FUNCTION_BLOCK DoorControl (* Basic Function Block Type *)
  (* Standard: 61499-2 *)
  (* Version 0.0, 6/17/2016, Andrei, nxtControl GmbH, Template *)
  PACKAGE Main;
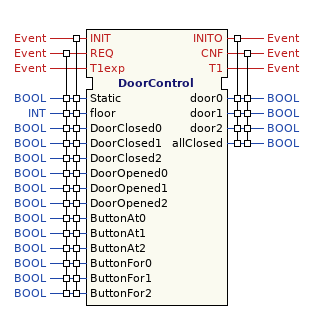
  EVENT_INPUT
    INIT WITH Static, floor, DoorClosed0, DoorClosed1, DoorClosed2, DoorOpened0, DoorOpened1, DoorOpened2, ButtonAt0, ButtonAt1, ButtonAt2, ButtonFor0, ButtonFor1, ButtonFor2; (* Initialization Request *)
    REQ WITH Static, floor, DoorClosed0, DoorClosed1, DoorClosed2, DoorOpened0, DoorOpened1, DoorOpened2, ButtonAt0, ButtonAt1, ButtonAt2, ButtonFor0, ButtonFor1, ButtonFor2; (* Normal Execution Request *)
    T1exp;
  END_EVENT
  EVENT_OUTPUT
    INITO WITH door0, door1, door2, allClosed; (* Initialization Confirm *)
    CNF WITH door0, door1, door2, allClosed; (* Execution Confirmation *)
    T1;
  END_EVENT
  VAR_INPUT
    Static : BOOL;
    floor : INT;
    DoorClosed0 : BOOL;
    DoorClosed1 : BOOL;
    DoorClosed2 : BOOL;
    DoorOpened0 : BOOL;
    DoorOpened1 : BOOL;
    DoorOpened2 : BOOL;
    ButtonAt0 : BOOL;
    ButtonAt1 : BOOL;
    ButtonAt2 : BOOL;
    ButtonFor0 : BOOL;
    ButtonFor1 : BOOL;
    ButtonFor2 : BOOL;
  END_VAR
  VAR_OUTPUT
    door0 : BOOL;
    door1 : BOOL;
    door2 : BOOL;
    allClosed : BOOL;
  END_VAR
  VAR
    doOpen0 : BOOL;
    doOpen1 : BOOL;
    doOpen2 : BOOL;
  END_VAR
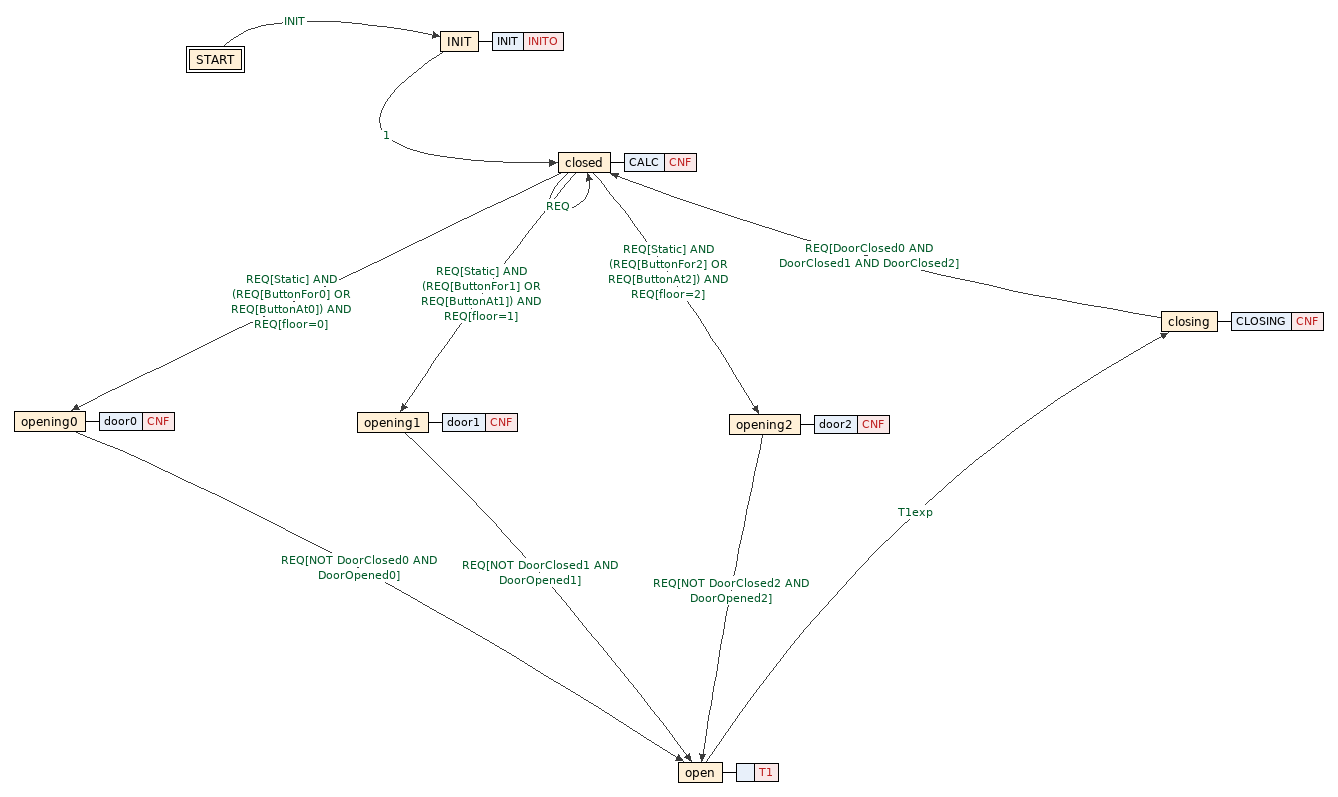
  EC_STATES
    START; (* Initial State *)
    INIT : INIT -> INITO;
    closed : CALC -> CNF;
    opening0 : door0 -> CNF;
    open : -> T1;
    closing : CLOSING -> CNF;
    opening1 : door1 -> CNF;
    opening2 : door2 -> CNF;
  END_STATES
  EC_TRANSITIONS
    START TO INIT := INIT;
    closed TO opening0 := REQ[Static] AND (REQ[ButtonFor0] OR REQ[ButtonAt0]) AND REQ[floor=0];
    open TO closing := T1exp;
    closing TO closed := REQ[DoorClosed0 AND DoorClosed1 AND DoorClosed2];
    opening0 TO open := REQ[NOT DoorClosed0 AND DoorOpened0];
    closed TO opening1 := REQ[Static] AND (REQ[ButtonFor1] OR REQ[ButtonAt1]) AND REQ[floor=1];
    opening1 TO open := REQ[NOT DoorClosed1 AND DoorOpened1];
    closed TO opening2 := REQ[Static] AND (REQ[ButtonFor2] OR REQ[ButtonAt2]) AND REQ[floor=2];
    opening2 TO open := REQ[NOT DoorClosed2 AND DoorOpened2];
    INIT TO closed := 1;
    closed TO closed := REQ;
  END_TRANSITIONS
  ALGORITHM INIT IN ST: (* Initialization algorithm *)
;
allClosed:=TRUE;
  END_ALGORITHM
  ALGORITHM door0 IN ST:
;
door0 := TRUE;
allClosed := FALSE;
  END_ALGORITHM
  ALGORITHM door1 IN ST:
;
door1 := TRUE;
allClosed := FALSE;
  END_ALGORITHM
  ALGORITHM door2 IN ST:
;
door2 := TRUE;
allClosed := FALSE;
  END_ALGORITHM
  ALGORITHM CALC IN ST:
;
allClosed:=TRUE;
door0 := FALSE;
door1 := FALSE;
door2 := FALSE;
  END_ALGORITHM
  ALGORITHM CLOSING IN ST:
;
door0:=FALSE;
door1:=FALSE;
door2:=FALSE;
  END_ALGORITHM
  ALGORITHM T1 IN ST:
;
T1exp := 0;
  END_ALGORITHM
END_FUNCTION_BLOCK
